FUNCTION_BLOCK IntegralController
  (* Standard: 61499-2 *)
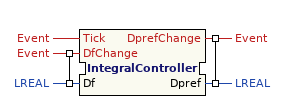
  EVENT_INPUT
    Tick;
    DfChange WITH Df;
  END_EVENT
  EVENT_OUTPUT
    DprefChange WITH Dpref;
  END_EVENT
  VAR_INPUT
    Df : LREAL;
  END_VAR
  VAR_OUTPUT
    Dpref : LREAL;
  END_VAR
  VAR
    StepSize : LREAL := 0.0001;
    Ki : LREAL := 0.6;
  END_VAR
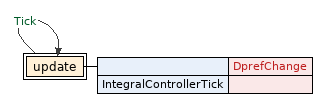
  EC_STATES
    update : -> DprefChange, IntegralControllerTick;
  END_STATES
  EC_TRANSITIONS
    update TO update := Tick;
  END_TRANSITIONS
  ALGORITHM IntegralControllerTick IN ST:
        Dpref := Dpref - (Ki*Df)*StepSize;
  END_ALGORITHM
END_FUNCTION_BLOCK
